// TwinCAT 3 PLC project Proj_sw01
// ProgramVersion: 3.1.4023.0
// libraries:
//   Tc2_Standard, * (Beckhoff Automation GmbH)
//   Tc2_System, * (Beckhoff Automation GmbH)
//   Tc3_Module, * (Beckhoff Automation GmbH)
//   VisuSymbols,3.5.10.0,System
// project tree:
//   / GlobalTextList.TcGTLO, PlcTask.TcTTO, Visualization Manager.TcVMO (not stored)
//   GVLs/ GVL_CONST.TcGVL, GVL_IO.TcGVL
//   POUs/ Fb_Counter.TcPOU, Fun_Counter.TcPOU, MAIN.TcPOU, Prg_Counter.TcPOU
//   VISUs/ Visualization.TcVIS
// real-time tasks:
//   TASK PlcTask: cycle T#10ms, priority 20, ADS port 350
//   TASK PlcTask1: cycle T#10ms, priority 21, ADS port 351
//   TASK PlcTask2: cycle T#10ms, priority 22, ADS port 352
// I/O:
//   DEVICE Device 1 (EtherCAT), AmsNetId 10.180.42.28.2.1
//     Term 1 (EK1200) [EK1200-5000 EtherCAT Power supply (2A E-Bus)]
//       Term 2 (EL1004) [EL1004 4Ch. Dig. Input 24V, 3ms]
//       Term 3 (EL2004) [EL2004 4Ch. Dig. Output 24V, 0.5A]
//       Term 4 (EL3004) [EL3004 4Ch. Ana. Input +/-10V]
//       Term 5 (EL4034) [EL4034 4Ch. Ana. Output +/-10V, 12bit]
//       Term 6 (EK1110) [EK1110 EtherCAT extension]
//     Term 7 (EK1100) [EK1100 EtherCAT Coupler (2A E-Bus)]
//       Term 8 (EL3311) [EL3311 1Ch. Ana. Input Thermocouple (TC)]
//       Term 9 (EL3255) [EL3255 5Ch. potentiometer measurement with sensor supply]
//       Box 10 (BK1250)
// variable links:
//   Proj_Ueb_sw01/Proj_Ueb_sw01 Instance <-> Device 1 (EtherCAT)/Term 1 (EK1200)/Term 2 (EL1004)
//     PlcTask Inputs/GVL_IO.DI_BtnBlue <-> Channel 2/Input
//     PlcTask Inputs/GVL_IO.DI_BtnYellow <-> Channel 1/Input
//   Proj_Ueb_sw01/Proj_Ueb_sw01 Instance <-> Device 1 (EtherCAT)/Term 1 (EK1200)/Term 3 (EL2004)
//     PlcTask Outputs/GVL_IO.DO_LampGreen <-> Channel 2/Output
//     PlcTask Outputs/GVL_IO.DO_LampRed <-> Channel 1/Output

CONFIGURATION Proj_sw01
    RESOURCE PLC ON TwinCAT3
        TASK PlcTask(INTERVAL := T#10ms, PRIORITY := 20);
        PROGRAM MAIN WITH PlcTask : MAIN;
    END_RESOURCE
END_CONFIGURATION

// ---- GVLs/GVL_CONST.TcGVL
{attribute 'qualified_only'}
VAR_GLOBAL CONSTANT
	analogOutputMaxVolt		: INT := 10;
	intMaxValue				: INT := 32767;
	samplingTime			: TIME := T#10S;
END_VAR

// ---- GVLs/GVL_IO.TcGVL
{attribute 'qualified_only'}
VAR_GLOBAL
	input1 : INT;
END_VAR

// ---- POUs/MAIN.TcPOU
PROGRAM MAIN
VAR
	count 				: INT := 0;
	i_CounterFun 		: INT := 0;
	i_CounterFunBlock	: INT := 0;
	i_CounterProgram	: INT := 0;
	
	fb_Count_obj1 		: Fb_Counter;
	
	timer1				: TON;
	timerPT				: TIME := T#10.0S;
	bTimerEnded			: BOOL := FALSE;
	bTimerIn			: BOOL;
END_VAR

// count := count + 1;

// count up with counter function
i_CounterFun := Fun_Counter(i_CounterFun); 



// count up with counter function block
fb_Count_obj1();   // call function block
i_CounterFunBlock := fb_Count_obj1.i_countOut;   // access variables



// count up using a program
Prg_Counter(i_countOut => i_CounterProgram);


// access global variable list
GVL_IO.input1;

// test with timer
timer1.IN := bTimerIn;  // pass input values
timer1.PT := timerPT;   
timer1();  // call fb
IF timer1.Q THEN
	bTimerEnded := TRUE;
END_IF

END_PROGRAM

// ---- POUs/Fb_Counter.TcPOU
FUNCTION_BLOCK Fb_Counter
VAR_INPUT
END_VAR
VAR_OUTPUT
	i_countOut			: INT;
END_VAR
VAR
	i_counter_save		: INT;
	i_countUp			: INT := 1;
END_VAR

i_counter_save := i_counter_save + i_countUp;
i_countOut := i_counter_save;

END_FUNCTION_BLOCK

// ---- POUs/Fun_Counter.TcPOU
FUNCTION Fun_Counter : INT
VAR_INPUT
	i_count_in 			: INT; 
END_VAR
VAR
	i_countUp 			: INT := 1;
END_VAR

Fun_Counter := i_count_in + i_countUp;

END_FUNCTION

// ---- POUs/Prg_Counter.TcPOU
PROGRAM Prg_Counter
VAR
	i_counter_save			: INT;
	i_countUp				: INT := 1;
END_VAR
VAR_OUTPUT
	i_countOut			: INT;
END_VAR

i_counter_save := i_counter_save + i_countUp;
i_countOut := i_counter_save;

END_PROGRAM

// ---- VISUs/Visualization.TcVIS
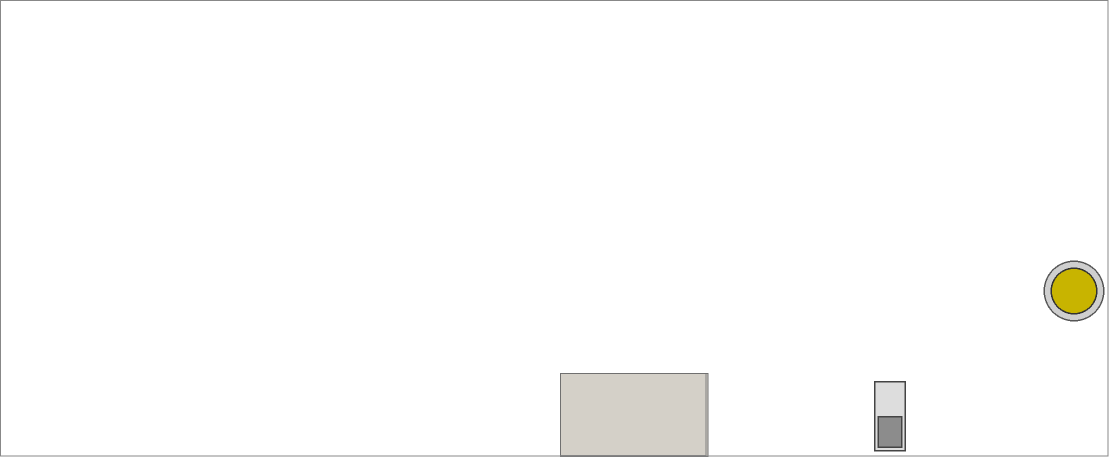
VISUALIZATION Visualization  // 1109x457
    Button (560,373 148x84)
    DipSwitch (855,381 70x70), variable: MAIN.bTimerIn, behaviour: TOGGLE, style: Switch-DipSwitch-Gray
    Lamp1 (1039,256 70x70), variable: MAIN.bTimerEnded, style: Lamp-Lamp1-Yellow
END_VISUALIZATION
